// TIA Portal V20 export
FUNCTION "fc_3" : Void   // FC2, LAD
{ S7_Optimized_Access := 'TRUE' }
// stored: SetENOAutomatically false
   VAR_TEMP
      Start : Bool;
      m_req : Bool;
      stop : Bool;
      Cond_1 : Bool;
      step_2 : Bool;
      step_1 : Bool;
      step_3 : Bool;
      fault : Bool;
      auto : Bool;
      man : Bool;
      CMD_Mot : Bool;
      "a" : Bool;
      y : Bool;
      aaaa : Bool;
   END_VAR
BEGIN

REGION Network 1: Set
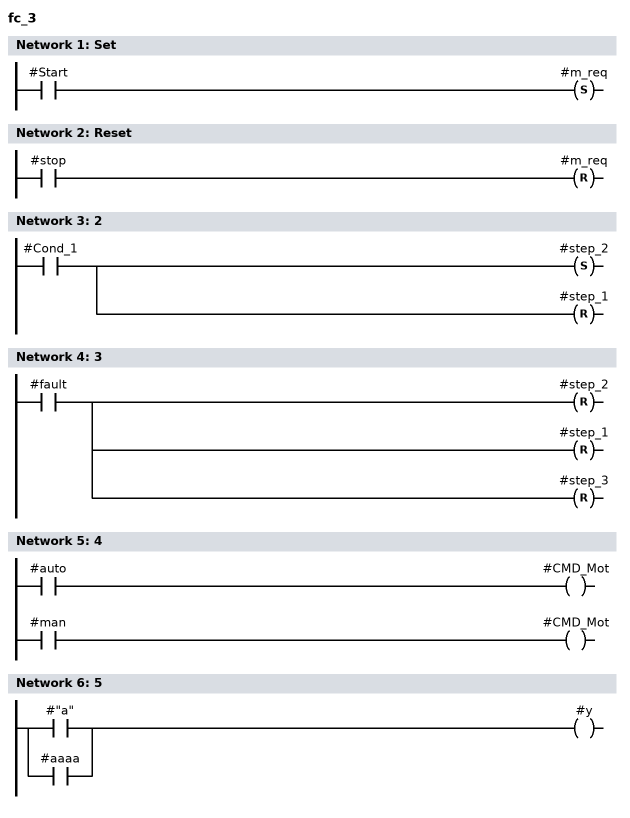
   RUNG wire#powerrail
      Contact( #Start )
      S_Coil( #m_req )
   END_RUNG
   // the same network as SCL:
   IF #Start THEN #m_req := TRUE; END_IF;
END_REGION

REGION Network 2: Reset
   RUNG wire#powerrail
      Contact( #stop )
      R_Coil( #m_req )
   END_RUNG
   // the same network as SCL:
   IF #stop THEN #m_req := FALSE; END_IF;
END_REGION

REGION Network 3: 2
   RUNG wire#powerrail
      Contact( #Cond_1 )
      wire#w1
      S_Coil( #step_2 )
   END_RUNG
   RUNG wire#w1
      R_Coil( #step_1 )
   END_RUNG
   // the same network as SCL:
   IF #Cond_1 THEN
       #step_2 := TRUE;
       #step_1 := FALSE;
   END_IF;
END_REGION

REGION Network 4: 3
   RUNG wire#powerrail
      Contact( #fault )
      wire#w1
      R_Coil( #step_2 )
   END_RUNG
   RUNG wire#w1
      R_Coil( #step_1 )
   END_RUNG
   RUNG wire#w1
      R_Coil( #step_3 )
   END_RUNG
   // the same network as SCL:
   IF #fault THEN
       #step_2 := FALSE;
       #step_1 := FALSE;
       #step_3 := FALSE;
   END_IF;
END_REGION

REGION Network 5: 4
   RUNG wire#powerrail
      Contact( #auto )
      Coil( #CMD_Mot )
   END_RUNG
   RUNG wire#powerrail
      Contact( #man )
      Coil( #CMD_Mot )
   END_RUNG
   // the same network as SCL:
   #CMD_Mot := #auto;
   #CMD_Mot := #man;
END_REGION

REGION Network 6: 5
   RUNG wire#powerrail
      Contact( #"a" )
      wire#w1
      Coil( #y )
   END_RUNG
   RUNG wire#powerrail
      Contact( #aaaa )
   END_RUNG wire#w1
   // the same network as SCL:
   #y := #"a" OR #aaaa;
END_REGION
END_FUNCTION
